FUNCTION_BLOCK Servo
VAR_INPUT
	HMI_MODE : BOOL;
END_VAR
VAR_OUTPUT
END_VAR
VAR
	fbPower 	: ARRAY [1..MAX_AXES] OF MC_POWER;
	fbReset 	: ARRAY [1..MAX_AXES] OF MC_RESET;
	fbHome		: ARRAY	[1..MAX_AXES] OF MC_HOME;
	fbMoveA 	: ARRAY [1..MAX_AXES] OF MC_MOVEABSOLUTE;
	fbMoveR 	: ARRAY [1..MAX_AXES] OF MC_MOVERELATIVE;
	fbJog		: ARRAY [1..MAX_AXES] OF MC_JOG;
	fbHalt	 	: ARRAY [1..MAX_AXES] OF MC_HALT;
	i			: INT;
END_VAR

IF HMI_MODE THEN 
	FOR i := 1 TO MAX_AXES BY 1 DO
		ACT_UpdateStatus();
		IF HmiToPlc[i].SERVO_OFF THEN
			ACT_Off();
		ELSIF HmiToPlc[i].SERVO_ON THEN 
			ACT_On();
		END_IF
		IF NOT HmiToPlc[i].SERVO_JOG_MODE THEN 
			Servo_Jog_Stop(i);
			IF HmiToPlc[i].SERVO_MOVE_ABS THEN
				ACT_MoveToPosition();
			END_IF
			IF HmiToPlc[i].SERVO_MOVE_REL THEN
				ACT_MoveByDistance();
			END_IF
		ELSE
			ACT_Jog();
		END_IF
	END_FOR
END_IF

ACTION ACT_On:
Servo_On(i, HmiToPlc[i].SERVO_ON_FW, HmiToPlc[i].SERVO_ON_BW, HmiToPlc[i].CONTROLLER_OVERRIDE);
END_ACTION

METHOD PUBLIC Servo_Home : ServoMotion_FunctionResult
VAR_INPUT
	INDEX : INT;
END_VAR
IF INDEX > MAX_AXES OR INDEX < 1 THEN 
	Servo_Home := ServoMotion_FunctionResult.MOTION_UNKNOWN_AXIS;
ELSE
	fbHome[INDEX](
		Axis:= AXIS[INDEX].AXIS, 
		Execute:= TRUE, 
		Position:= 0, 
		HomingMode:= MC_DefaultHoming, 
		bCalibrationCam:= AXIS[INDEX].HOME_CALIBRATION );
	IF fbHome[INDEX].Error THEN
		fbHome[INDEX](
			Axis:= AXIS[INDEX].AXIS, 
			Execute:= FALSE );
		Servo_Home := ServoMotion_FunctionResult.MOTION_ERROR;
	ELSIF fbHome[INDEX].CommandAborted THEN
		fbHome[INDEX](
			Axis:= AXIS[INDEX].AXIS, 
			Execute:= FALSE );
		Servo_Home := ServoMotion_FunctionResult.MOTION_COMMAND_ABORTED;
	ELSIF fbHome[INDEX].Done THEN
		fbHome[INDEX](
			Axis:= AXIS[INDEX].AXIS, 
			Execute:= FALSE );
		Servo_Home := ServoMotion_FunctionResult.MOTION_OK;
	ELSE
		Servo_Home := ServoMotion_FunctionResult.MOTION_BUSY;
	END_IF
END_IF
END_METHOD

METHOD PUBLIC Servo_Jog_Stop : ServoMotion_FunctionResult
VAR_INPUT
	INDEX : INT;
END_VAR
fbJog[INDEX](
	Axis:= AXIS[INDEX].AXIS, 
	JogForward:= FALSE, 
	JogBackwards:= FALSE );
IF fbJog[INDEX].Error THEN 
	Servo_Jog_Stop := ServoMotion_FunctionResult.MOTION_ERROR;
ELSE
	Servo_Jog_Stop := ServoMotion_FunctionResult.MOTION_OK;
END_IF
END_METHOD

METHOD PUBLIC Servo_Off : ServoMotion_FunctionResult
VAR_INPUT
	INDEX : INT;
END_VAR
IF INDEX > MAX_AXES OR INDEX < 1 THEN 
	Servo_Off := ServoMotion_FunctionResult.MOTION_UNKNOWN_AXIS;
ELSE
	fbPower[INDEX](
		Axis:= AXIS[INDEX].AXIS, 
		Enable:= FALSE, 
		Enable_Positive:= FALSE, 
		Enable_Negative:= FALSE, 
		Override:= 0 );
	IF fbPower[INDEX].Error THEN
		Servo_Off := ServoMotion_FunctionResult.MOTION_ERROR;
	ELSIF NOT fbPower[INDEX].Status THEN
		Servo_Off := ServoMotion_FunctionResult.MOTION_OK;
	ELSE
		Servo_Off := ServoMotion_FunctionResult.MOTION_BUSY;
	END_IF
END_IF
END_METHOD

ACTION ACT_MoveToPosition:
CASE Servo_MoveToPosition(i,HmiToPlc[i].TARGET_POSITION,HmiToPlc[i].TARGET_VELOCITY,HmiToPlc[i].TARGET_ACCELERATION,HmiToPlc[i].TARGET_DECELERATION,HmiToPlc[i].TARGET_JERK) OF
ServoMotion_FunctionResult.MOTION_UNKNOWN_AXIS:
	;
ServoMotion_FunctionResult.MOTION_COMMAND_ABORTED: 
	;
ServoMotion_FunctionResult.MOTION_ERROR:
	;
ServoMotion_FunctionResult.MOTION_BUSY: 
	;
ServoMotion_FunctionResult.MOTION_OK:
	;
END_CASE
END_ACTION

PROPERTY PUBLIC AXIS_COUNT : INT
GET
AXIS_COUNT := MAX_AXES;
END_GET
END_PROPERTY

METHOD PUBLIC Servo_MoveToPosition : ServoMotion_FunctionResult
VAR_INPUT
	INDEX 			: INT;
	POSITION		: LREAL;
	VELOCITY		: LREAL;
	ACCELERATION	: LREAL;
	DECELERATION	: LREAL;
	JERK			: LREAL;
END_VAR
IF INDEX > MAX_AXES OR INDEX < 1 AND VELOCITY <= 0 THEN 
	Servo_MoveToPosition := ServoMotion_FunctionResult.MOTION_UNKNOWN_AXIS;
ELSE
	fbMoveA[INDEX](
		Axis:= AXIS[INDEX].AXIS, 
		Execute:= TRUE, 
		Position:= POSITION, 
		Velocity:= VELOCITY, 
		Acceleration:= ACCELERATION, 
		Deceleration:= DECELERATION, 
		Jerk:= JERK );
	IF fbMoveA[INDEX].Error THEN
		fbMoveA[INDEX](
			Axis:= AXIS[INDEX].AXIS, 
			Execute:= FALSE );
		Servo_MoveToPosition := ServoMotion_FunctionResult.MOTION_ERROR;
	ELSIF fbMoveA[INDEX].CommandAborted THEN
		fbMoveA[INDEX](
			Axis:= AXIS[INDEX].AXIS, 
			Execute:= FALSE );
		Servo_MoveToPosition := ServoMotion_FunctionResult.MOTION_COMMAND_ABORTED;
	ELSIF fbMoveA[INDEX].Done THEN
		fbMoveA[INDEX](
			Axis:= AXIS[INDEX].AXIS, 
			Execute:= FALSE );
		Servo_MoveToPosition := ServoMotion_FunctionResult.MOTION_OK;
	ELSE
		Servo_MoveToPosition := ServoMotion_FunctionResult.MOTION_BUSY;
	END_IF
END_IF
END_METHOD

ACTION ACT_Off:
Servo_Off(i);
END_ACTION

METHOD PUBLIC Servo_Halt : ServoMotion_FunctionResult
VAR_INPUT
	INDEX : INT;
END_VAR
IF INDEX > MAX_AXES OR INDEX < 1 THEN 
	Servo_Halt := ServoMotion_FunctionResult.MOTION_UNKNOWN_AXIS;
ELSE
	fbHalt[INDEX](
		Axis:= AXIS[INDEX].AXIS, 
		Execute:= TRUE );
	fbMoveA[INDEX](
		Axis:= AXIS[INDEX].AXIS, 
		Execute:= FALSE );
	fbMoveR[INDEX](
		Axis:= AXIS[INDEX].AXIS, 
		Execute:= FALSE );
	IF fbHalt[INDEX].Error THEN
		fbHalt[INDEX](
			Axis:= AXIS[INDEX].AXIS, 
			Execute:= FALSE );
		Servo_Halt := ServoMotion_FunctionResult.MOTION_ERROR;
	ELSIF fbHalt[INDEX].CommandAborted THEN
		fbHalt[INDEX](
			Axis:= AXIS[INDEX].AXIS, 
			Execute:= FALSE );
		Servo_Halt := ServoMotion_FunctionResult.MOTION_COMMAND_ABORTED;
	ELSIF fbHalt[INDEX].Done THEN
		fbHalt[INDEX](
			Axis:= AXIS[INDEX].AXIS, 
			Execute:= FALSE );
		Servo_Halt := ServoMotion_FunctionResult.MOTION_OK;
	ELSE
		Servo_Halt := ServoMotion_FunctionResult.MOTION_BUSY;
	END_IF
END_IF
END_METHOD

ACTION ACT_MoveByDistance:
CASE Servo_MoveByDistance(i,HmiToPlc[i].TARGET_POSITION,HmiToPlc[i].TARGET_VELOCITY,HmiToPlc[i].TARGET_ACCELERATION,HmiToPlc[i].TARGET_DECELERATION,HmiToPlc[i].TARGET_JERK) OF
ServoMotion_FunctionResult.MOTION_UNKNOWN_AXIS:
	;
ServoMotion_FunctionResult.MOTION_COMMAND_ABORTED: 
	;
ServoMotion_FunctionResult.MOTION_ERROR:
	;
ServoMotion_FunctionResult.MOTION_BUSY: 
	;
ServoMotion_FunctionResult.MOTION_OK:
	;
END_CASE
END_ACTION

METHOD PUBLIC Servo_Jog_Start : ServoMotion_FunctionResult
VAR_INPUT
	INDEX		: INT;
	REVERSE		: BOOL := FALSE;
	FAST_MODE	: BOOL := FALSE;
END_VAR
IF FAST_MODE THEN 
	fbJog[INDEX].Mode := MC_JOGMODE_STANDARD_FAST;
ELSE
	fbJog[INDEX].Mode := MC_JOGMODE_STANDARD_SLOW;
END_IF

fbJog[INDEX](
	Axis:= AXIS[INDEX].AXIS, 
	JogForward:= NOT REVERSE, 
	JogBackwards:= REVERSE );
IF fbJog[INDEX].Error THEN 
	Servo_Jog_Start := ServoMotion_FunctionResult.MOTION_ERROR;
ELSIF AXIS[INDEX].AXIS.Status.Moving THEN 
	Servo_Jog_Start := ServoMotion_FunctionResult.MOTION_OK;
END_IF
END_METHOD

PROPERTY AxisGroup_Count : INT
GET
AXISGROUP_Count := MAX_AXIS_GROUPS;
END_GET
END_PROPERTY

ACTION ACT_Reset:
IF Servo_Reset(i) = ServoMotion_FunctionResult.MOTION_OK THEN
	HmiToPlc[i].SERVO_RESET := FALSE;
END_IF
END_ACTION

METHOD PUBLIC Servo_MoveByDistance : ServoMotion_FunctionResult
VAR_INPUT
	INDEX 			: INT;
	DISTANCE 		: LREAL;
	VELOCITY 		: LREAL;
	ACCELERATION 	: LREAL;
	DECELERATION 	: LREAL;
	JERK 			: LREAL;
END_VAR
IF INDEX > MAX_AXES OR INDEX < 1 AND VELOCITY <= 0 THEN 
	Servo_MoveByDistance := ServoMotion_FunctionResult.MOTION_UNKNOWN_AXIS;
ELSE
	fbMoveR[INDEX](
		Axis:= AXIS[INDEX].AXIS, 
		Execute:= TRUE, 
		Distance:= DISTANCE, 
		Velocity:= VELOCITY, 
		Acceleration:= ACCELERATION, 
		Deceleration:= DECELERATION, 
		Jerk:= JERK );
	IF fbMoveR[INDEX].Error THEN
		fbMoveR[INDEX](
			Axis:= AXIS[INDEX].AXIS, 
			Execute:= FALSE );
		Servo_MoveByDistance := ServoMotion_FunctionResult.MOTION_ERROR;
	ELSIF fbMoveR[INDEX].CommandAborted THEN
		fbMoveR[INDEX](
			Axis:= AXIS[INDEX].AXIS, 
			Execute:= FALSE );
		Servo_MoveByDistance := ServoMotion_FunctionResult.MOTION_COMMAND_ABORTED;
	ELSIF fbMoveR[INDEX].Done THEN
		fbMoveR[INDEX](
			Axis:= AXIS[INDEX].AXIS, 
			Execute:= FALSE );
		Servo_MoveByDistance := ServoMotion_FunctionResult.MOTION_OK;
	ELSE
		Servo_MoveByDistance := ServoMotion_FunctionResult.MOTION_BUSY;
	END_IF
END_IF
END_METHOD

ACTION ACT_Jog:
IF HmiToPlc[i].SERVO_JOG_FW_FAST THEN
	Servo_Jog_Start(i, FALSE, TRUE);
ELSIF HmiToPlc[i].SERVO_JOG_FW_SLOW THEN
	Servo_Jog_Start(i, FALSE, FALSE);
ELSIF HmiToPlc[i].SERVO_JOG_BW_FAST THEN
	Servo_Jog_Start(i, TRUE, TRUE);
ELSIF HmiToPlc[i].SERVO_JOG_BW_SLOW THEN
	Servo_Jog_Start(i, TRUE, FALSE);
ELSE
	Servo_Jog_Stop(i);
END_IF
END_ACTION

METHOD Servo_On : ServoMotion_FunctionResult
VAR_INPUT
	INDEX : INT;
	ENABLE_FW 	: BOOL;
	ENABLE_BW	: BOOL;
	OVERRIDE	: LREAL;
END_VAR
IF INDEX > MAX_AXES OR INDEX < 1 THEN 
	Servo_On := ServoMotion_FunctionResult.MOTION_UNKNOWN_AXIS;
ELSE
	fbPower[INDEX](
		Axis:= AXIS[INDEX].AXIS, 
		Enable:= TRUE, 
		Enable_Positive:= ENABLE_FW, 
		Enable_Negative:= ENABLE_BW, 
		Override:= OVERRIDE );
	IF fbPower[INDEX].Error THEN
		Servo_On := ServoMotion_FunctionResult.MOTION_ERROR;
	ELSIF fbPower[INDEX].Status THEN
		Servo_On := ServoMotion_FunctionResult.MOTION_OK;
	ELSE
		Servo_On := ServoMotion_FunctionResult.MOTION_BUSY;
	END_IF
END_IF
END_METHOD

METHOD PUBLIC Servo_Reset : ServoMotion_FunctionResult
VAR_INPUT
	INDEX :INT;
END_VAR
IF INDEX > MAX_AXES OR INDEX < 1 THEN 
	Servo_Reset := ServoMotion_FunctionResult.MOTION_UNKNOWN_AXIS;
ELSE
	fbReset[INDEX](
		Axis:= AXIS[INDEX].AXIS, 
		Execute:= TRUE );
	IF fbReset[INDEX].Error THEN
		fbReset[INDEX](
			Axis:= AXIS[INDEX].AXIS, 
			Execute:= FALSE );
		Servo_Reset := ServoMotion_FunctionResult.MOTION_ERROR;
	ELSIF fbReset[INDEX].Done THEN
		fbReset[INDEX](
			Axis:= AXIS[INDEX].AXIS, 
			Execute:= FALSE );
		Servo_Reset := ServoMotion_FunctionResult.MOTION_OK;
	ELSE
		Servo_Reset := ServoMotion_FunctionResult.MOTION_BUSY;
	END_IF
END_IF
END_METHOD

ACTION ACT_UpdateStatus:
AXIS[i].AXIS.ReadStatus();
PlcToHmi[i].actPos	:= AXIS[i].AXIS.NcToPlc.ActPos;
PlcToHmi[i].actVelo := AXIS[i].AXIS.NcToPlc.ActVelo;
PlcToHmi[i].setPos	:= AXIS[i].AXIS.NcToPlc.SetPos;
PlcToHmi[i].setVelo := AXIS[i].AXIS.NcToPlc.SetVelo;
PlcToHmi[i].controller_override := fbPower[i].Override;
PlcToHmi[i].hasError := AXIS[i].AXIS.Status.Error;
PlcToHmi[i].ErrorID := AXIS[i].AXIS.Status.ErrorID;
PlcToHmi[i].isBwDisabled := NOT fbPower[i].Enable_Negative;
PlcToHmi[i].isFwDisabled := NOT fbPower[i].Enable_Positive;
PlcToHmi[i].isCalibrated := AXIS[i].AXIS.Status.Homed;
PlcToHmi[i].isDisabled := AXIS[i].AXIS.Status.Disabled;
PlcToHmi[i].isInRange := AXIS[i].AXIS.Status.InPositionArea;
PlcToHmi[i].isInTarget := AXIS[i].AXIS.Status.InTargetPosition;
PlcToHmi[i].isNegativeDirection := AXIS[i].AXIS.Status.NegativeDirection;
PlcToHmi[i].isNotMoving := AXIS[i].AXIS.Status.NotMoving;
PlcToHmi[i].isPositiveDirection := AXIS[i].AXIS.Status.PositiveDirection;
END_ACTION

END_FUNCTION_BLOCK

(* stored: Version 1.1.0.1, ProductVersion 3.1.0.36
   POU Servo: Id {55b379f4-f721-4632-9623-aca35a4ff0b7}, SpecialFunc None
   Folder HMI Actions: Id {a81ee722-85c9-42c1-866f-016e6d583404}
   Action ACT_On: Id {055125fe-25ee-4a7a-b050-73eb03772677}
   Method Servo_Home: Id {177da0d7-0e75-4752-b88f-e867267c266c}
   Method Servo_Jog_Stop: Id {1f8fc547-a813-4b5f-93fa-9fae40058f6f}
   Method Servo_Off: Id {2b7678fb-5114-4046-a0d3-11070b4fbd98}
   Action ACT_MoveToPosition: Id {40847845-e28a-467f-8c2b-007d9c73cf9b}
   Property AXIS_COUNT: Id {459cb5a1-6ab5-4653-9f1f-4943f3702408}
   Get Get: Id {9be2d030-51e7-4e34-80b7-5636315565bf}
   Method Servo_MoveToPosition: Id {4b4bad53-575d-4566-847b-5df400e707ed}
   Action ACT_Off: Id {5bdb5604-b204-4401-92fa-0d357435d921}
   Method Servo_Halt: Id {6989ff12-21aa-479d-ad23-23232d5ecada}
   Action ACT_MoveByDistance: Id {7d58b39d-b312-4669-b3d1-c2d6a9066f91}
   Method Servo_Jog_Start: Id {857d1325-691b-4e71-89f9-5cc1b73fa800}
   Property AxisGroup_Count: Id {9f93d7b8-c6c0-420b-b549-25dfd1d07367}
   Get Get: Id {6c4c1b83-d2cd-4270-b6f4-b61728b59c66}
   Action ACT_Reset: Id {a7a36296-4bd3-4c04-bfcc-ad271ca28fe6}
   Method Servo_MoveByDistance: Id {b7b49934-4930-4ea2-b772-a6e74f151dd6}
   Action ACT_Jog: Id {cc0383b4-9148-4bf0-9c5a-f7313178b54b}
   Method Servo_On: Id {d7c9e2a6-ab50-4fb9-bb77-ce0d39e7247b}
   Method Servo_Reset: Id {e126d8bd-3570-40c3-9468-28dd8d3340a4}
   Action ACT_UpdateStatus: Id {fc19d8f7-7aab-443d-a6b0-6c271a3d11f7} *)
